{attribute 'GeneratedUsingTerminal: EK1122-0000-0018'}
{attribute addProperty BoxType "EK1122-0000-0018"}
{attribute addProperty Id "Beckhoff_EJ9xxxsub_EK1100EK1100_AB5A94672"}
{attribute addProperty CRC "640976645"}
{attribute addProperty Size "2"}
TYPE Beckhoff_EJ9xxxEK1122_26348705 EXTENDS EK1122_AB5A9467 :
STRUCT
	{attribute addProperty Name "Beckhoff_EJ9xxxsub_EK1100"}
	{attribute addProperty PreviousPort "Beckhoff EJ9xxxEK1122 : D"}
	Beckhoff_EJ9xxxsub_EK1100 : EK1100_AB5A9467;
END_STRUCT
END_TYPE

(* stored: Version 1.2.0.0, ProductVersion 3.1.4024.9
   DUT Beckhoff_EJ9xxxEK1122_26348705: Id {ffba4b58-9176-452b-a471-5d8d0229e7f0} *)
